(* CoDeSys 2.3 export: PROC_ERR_PWM.EXP *)

(* POU 60_Error handling/Process Errors/proc_Err_PWM, ST *)
PROGRAM proc_Err_PWM
VAR
	ProcessErr1_fb: 			handleError;
	ProcessErr2_fb: 			handleError;
	ProcessErr3_fb: 			handleError;
	ProcessErr4_fb: 			handleError;
	ProcessErr5_fb: 			handleError;
	ProcessErr6_fb: 			handleError;
	ProcessErr7_fb: 			handleError;
	ProcessErr8_fb: 			handleError;

	ProcessErr9_fb: 			handleError;
	ProcessErr10_fb: 			handleError;
	ProcessErr11_fb: 			handleError;
	ProcessErr12_fb: 			handleError;



END_VAR
;
END_PROGRAM
